FUNCTION_BLOCK FB_InkCirculation EXTENDS FB_BaseInk IMPLEMENTS I_SleepObserver, I_EmergencyObserver

VAR_INPUT
  InActValue                 AT %I* : INT;                      (*Actual value*)
  IbActValueWcState          AT %I* : BOOL;                     (*EM3701 pressure WcState*)
  IbInkLevelReachedBack      AT %I* : BOOL;                     (*HT back level reached*)

  iPurgeController                  : I_Purge;
  iMencController                   : I_AirVolume;

  IbEnable                          : BOOL;                     (*Enable function*)
  IbAxisMovement                    : BOOL;                     (*Axis movement*)
  IbHeadertankOk                    : BOOL;                     (*Headertank ok*)
  IbPHTempOk                        : BOOL;                     (*Printhead temperature ok*)
END_VAR

VAR_OUTPUT
  ObHtCloseInkConnectionValve       : BOOL;                     (*HT: close ink connection valve front to back*)
  ObHtCloseMencConnectionValve      : BOOL;                     (*HT back: close menc connection valve*)
  ObValveActivation                 : BOOL;                     (*HT: valve activation*)
  ObPumpActivation                  : BOOL;                     (*HT: pump activation*)
END_VAR

VAR
  _sName                            : STRING;                   (*Block name*)

  _bEStop                           : BOOL := FALSE;            (*EStop active*)
  _bSleep                           : BOOL := FALSE;            (*Sleep active*)
  bCheckParameterError01            : BOOL := FALSE;            (*CheckParameter: error 01 reported*)
  bLevelError                       : BOOL := FALSE;            (*HT back level error*)
  bCirculationActive                : BOOL;                     (*Circulation active*)
  bConditionsMet                    : BOOL;                     (*Conditions met*)
  bPumpActivation                   : BOOL;                     (*HT: pump activation*)
  fbTpPumpOn                        : TP;                       (*HT: pump activation on*)
  tPumpOnTime                       : TIME;                     (*HT: pump activation on*)
  fbTpPumpWait                      : TP;                       (*HT: pump activation wait*)
  tPumpWaitTime                     : TIME;                     (*HT: pump activation wait*)
  bResetErrorCounter                : BOOL;                     (*Reset HT back level error counter*)

  fbTonSubMencOK                    : TON;                      (*Sub menc pressure ok*)
  fbTonNoMovement                   : TON;                      (*No axis movement active*)
  fbTonResumeCirculation            : TON;                      (*Resume circulation after level error*)

  fSubMencActValue                  : LREAL;                    (*HT: actual pressure of back side*)
  fSubMencTargetValue               : LREAL;                    (*HT: target pressure of back side*)
END_VAR

VAR PERSISTENT
  tRSubMencOk                       : TIME := T#5S;             (*Supervision time for sub menc ok*)
  tRNoMovement                      : TIME := T#1M;             (*Supervision time axis movement*)
  tRResumeCirculation               : TIME := T#1M;             (*Resume circulation after level error*)
  tRPumpDutyCycleFrequency          : TIME := T#100MS;          (*Frequency for duty cycle of pump*)
  nRPumpDutyCycle                   : UINT := 30;               (*Duty cycle of pump*)

  fRConvAdsToLocal                  : LREAL := 10.0;            (*Factor to convert from ADS to local*)
  fRSubMencDeltaP                   : LREAL := -2.5;            (*HT: delta pressure of sub menc on back side*)
  fRSubMencHysteresisP              : LREAL :=  0.5;            (*HT: hysteresis pressure*)
  fRSubMencCorrectionP              : LREAL :=  0.0;            (*HT: correction pressure*)

  nRErrorCounter                    : UINT := 0;                (*HT back level error counter*)
END_VAR

(*--- check parameter -------------------*)
IF NOT mCheckParameter() THEN RETURN; END_IF

(*HT back error*)
IF bCirculationActive AND IbInkLevelReachedBack THEN
  bLevelError    := TRUE;
  nRErrorCounter := nRErrorCounter + 1;
END_IF
fbTonResumeCirculation(IN := bLevelError, PT := tRResumeCirculation);
IF fbTonResumeCirculation.Q THEN
  bLevelError    := FALSE;
END_IF
IF bResetErrorCounter THEN
  nRErrorCounter := 0;
END_IF

fbTonSubMencOK (IN := (iMencController.pErrorCode = 0), PT := tRSubMencOk);
fbTonNoMovement(IN := NOT IbAxisMovement, PT := tRNoMovement);

fSubMencActValue    := INT_TO_LREAL(InActValue) / fRConvAdsToLocal;
fSubMencActValue    := fSubMencActValue + fRSubMencCorrectionP;
fSubMencTargetValue := iMencController.pPressure + fRSubMencDeltaP;

bConditionsMet :=     NOT IbActValueWcState
                  AND NOT _bEStop
                  AND NOT _bSleep
                  AND NOT IbInkLevelReachedBack
                  AND NOT bLevelError
                  AND NOT iPurgeController.pPurgeBusy
                  AND fbTonSubMencOK.Q
                  AND fbTonNoMovement.Q
                  AND IbHeadertankOk
                  AND IbPHTempOk
                  AND (fRSubMencDeltaP <> 0);

IF IbEnable AND bConditionsMet THEN
  bCirculationActive           := TRUE;
  ObHtCloseInkConnectionValve  := TRUE;
  ObHtCloseMencConnectionValve := TRUE;
  ObValveActivation            := TRUE;

  IF fSubMencActValue >= (fSubMencTargetValue + fRSubMencHysteresisP) THEN
    bPumpActivation := TRUE;
  END_IF
  IF fSubMencActValue <= (fSubMencTargetValue - fRSubMencHysteresisP) THEN
    bPumpActivation := FALSE;
  END_IF
ELSE  
  bCirculationActive           := FALSE;
  ObHtCloseInkConnectionValve  := FALSE;
  ObHtCloseMencConnectionValve := FALSE;
  ObValveActivation            := FALSE;
  bPumpActivation              := FALSE;
END_IF

(*Pump is activated with a variable duty cycle*)
tPumpOnTime   := DINT_TO_TIME((TIME_TO_DINT(tRPumpDutyCycleFrequency) * nRPumpDutyCycle) / 100);
tPumpWaitTime := DINT_TO_TIME((TIME_TO_DINT(tRPumpDutyCycleFrequency) * (100 - nRPumpDutyCycle)) / 100);
IF bPumpActivation THEN
  IF (nRPumpDutyCycle = 0) THEN
    ObPumpActivation := FALSE;
  ELSIF (nRPumpDutyCycle = 100) THEN
    ObPumpActivation := TRUE;
  ELSE
    fbTpPumpOn  (IN := NOT fbTpPumpWait.Q, PT := tPumpOnTime);
    fbTpPumpWait(IN := NOT fbTpPumpOn.Q  , PT := tPumpWaitTime);
  
    ObPumpActivation := fbTpPumpOn.Q;
  END_IF
ELSE
  fbTpPumpOn  (IN := FALSE);
  fbTpPumpWait(IN := FALSE);

  ObPumpActivation := FALSE;
END_IF

(*
  Check if all necessary variables are properly defined 
  - check if initialized
  - crash prevention!
*)
METHOD PRIVATE mCheckParameter : BOOL
IF (iPurgeController = 0) OR (iMencController = 0) THEN
  IF NOT bCheckParameterError01 THEN
    bCheckParameterError01 := TRUE;
    F_Report_Error(Report_Error_0Pointer);
  END_IF
  RETURN;
END_IF

mCheckParameter := TRUE; // all params ok
END_METHOD

METHOD mEmergencyUpdate
VAR_INPUT
	(*updated estop value TRUE = active*)
	bEStop	: BOOL;
END_VAR
_bEStop := bEStop;
END_METHOD

METHOD mSleepUpdate
VAR_INPUT
	(*updated sleep value TRUE = active*)
	bSleep	: BOOL;
END_VAR
_bSleep := bSleep;
END_METHOD

PROPERTY pName : STRING
SET
_sName := pName;
END_SET
END_PROPERTY

END_FUNCTION_BLOCK

(* stored: Version 1.1.0.1, ProductVersion 3.1.4024.11
   POU FB_InkCirculation: Id {60fff47b-915a-467a-9d62-9ebebbdf69ec}, SpecialFunc None
   Folder I_EmergencyObserver: Id {701194f4-da54-4e49-b47a-e21921119b4a}
   Folder I_SleepObserver: Id {1432cc03-7a96-4e1d-943e-d3d13817efe0}
   Method mCheckParameter: Id {484d4591-ac94-4d9d-ae00-0376398b1d80}
   Method mEmergencyUpdate: Id {46eb74cf-352d-4061-ac84-a2c24f18ce2b}
   Method mSleepUpdate: Id {6c063da7-a206-4a4d-91d3-7d17c61d638f}
   Property pName: Id {85d9f1e5-00c8-4693-bb26-b096ca7df051}
   Set Set: Id {db53bc8c-1af9-422a-90f1-c40afc967e04} *)
